PROGRAM MAIN
VAR_INPUT
	xInit			:BOOL:=TRUE;
END_VAR
VAR
	fbRef : ReferenceBlock;
END_VAR

IF xInit THEN
	xInit:=FALSE;
	fbRef();
END_IF

END_PROGRAM

(* stored: Version 1.1.0.1, ProductVersion 3.1.4024.10
   POU MAIN: Id {5f2e6d7d-97ea-4e54-81a5-1d341896552d}, SpecialFunc None *)
